FUNCTION_BLOCK Sensor_Trigger implements O_Sensor
VAR
	bOutput AT %Q* : BOOL;
END_VAR

PROPERTY isTriggered : BOOL
GET
isTriggered:=bOutput;
END_GET
END_PROPERTY

END_FUNCTION_BLOCK

(* stored: Version 1.1.0.1, ProductVersion 3.1.4024.12
   POU Sensor_Trigger: Id {989a519e-157f-43a1-bd04-99f835a50575}, SpecialFunc None
   Property isTriggered: Id {d41d1f0e-91df-4526-9abe-c5b6a9542aa8}
   Get Get: Id {522e1a2e-332e-482f-8b7b-83941e2bb972} *)
